Staubli VAL3: RosSimpleMsg.dtx

public Header header
  [0]
    num nMsgType
    num nCommType
    num nReplyCode
    num nData[12]
public Prefix prefix
  [0]
    num nLength
    num nData[4]
